// SIMATIC S7-200 project (STEP 7-Micro/WIN), CPU 226 REL 02.00

SYMBOL_TABLE USR1
d1               VD100    // Paper Core
HC               VD0      // Hi Speed Count
HCA              VD150    // Mill Roll Hi speed counter O.S
HCB              VD160    // Mill Roll Hi speed counter D.S
D                VD104    // Diameter
D2               VD108    // Diameter Limit
OUT              VD4      // Hi Speed Count Value
nip              VD112    // Nip
L                VD130    // Web Width
A                VD138    // Nip Setting
nipd             VD116    // Nip display
P                VD120    // Hydraulic press
V                VD204    // Analog out put
DC               AQW0     // 0-10VDC
S3               I0.2     // Paper to lead
S6               I0.5     // Rider roll slow up limit
S9               I1.0     // Lower cradle up limit
S10              I1.1     // Lower cradle down limit
S11              I1.2     // Lower cradle slow down limit
S12              I1.3     // Core chuck (D)
S13              I1.4     // Core chuck p.sw
CS1              I1.5     // Hydraulic pump
PB1              I1.6     // Hydraulic pump on
PB2              I1.7     // Hydraulic pump off
PB3              I2.0     // Trim removal fan ON
PB4              I2.1     // Trim removal fan OFF
PB5              I2.2     // Roll enjctor eject
PB6              I2.3     // Roll ejector return
PB7              I2.4     // Lead roll ON
PB8              I2.5     // Lead roll OFF
PB9              I2.6     // Web tail up
PB10             I2.7     // Web tail down
PB11             I3.0     // Core chuck lift up
PB12             I3.1     // Core chuck lift work
PB13             I3.2     // Core chuck lift down
PB14             I3.3     // Core chuck load
PB15             I3.4     // Core chuck open
PB16             I3.5     // Rder roll up
PB17             I3.6     // Rider roll work
PB18             I3.7     // Rder roll down
PB19             I4.0     // Lower cradle up
PB20             I4.1     // Lower cradle down
PB21             I4.2     // Clutch close
PB22             I4.3     // Auto roll ejector
PB23             I4.4     // Unwinder roll hold
PB24             I4.5     // Unwinder roll release
SP7              I4.6     // sp
SP8              I4.7     // sp
PB27             I5.0     // Lead roll up
PB28             I5.1     // Lead roll down
S14              I5.2     // Water Sensor(oper.side)
S15              I5.3     // Water Sensor(driver.side)
S16              I5.4     // Clutch open limit
S17              I5.5     // Clutch close limit
PB29             I5.6     // Crawl ON
PB30             I5.7     // Crawl  OFF
PB31             I6.0     // Trim ON
PB32             I6.1     // Trim OFF
PB33             I6.2     // Slitter ON
PB34             I6.3     // Slitter OFF
PB35             I6.4     // Blow ON
PB36             I6.5     // Blow OFF
OL1              I6.6     // Trim removal fan OL
OL2A             I6.7     // Hydraulic pump A OL
OL2B             I7.0     // Hydraulic pump B OL
OL3              I7.1     // Lead roll OL
EMG              I7.2     // Emergency
S18              I7.3     // Roll ejector middle limit
ABB1             I7.4     // TOSHIBA RUN
ABB2             I7.5     // TOSHIBA 0 speed
ABB3             I7.6     // TOSHIBA crawl
ABB4             I7.7     // TOSHIBA fault
ABB5             I8.0     // TOSHIBA unwinder brake
ABB6             I8.1     // TOSHIBA lead roll brake
ABB7             I8.2     // TOSHIBA drum brake
ABB8             I8.3     // TOSHIBA warning
S1               I8.4     // Roll ejector forware limit
S2               I8.5     // Roll ejector backware limit
S19              I8.6     // Lead roll motor up limit
S20              I8.7     // Lead roll motor down limit
S13A             I9.0     // Core chuck backward limit
SP4              I9.1     // Mill Roll up-down Motor Over Load O.S
SP5              I9.2     // Mill Roll up-down Motor Over Load D.S
OL8              I9.3     // Mill Roll Move Motor Over Load O.S
S23              I9.4     // Sheed cutter forward limit
S24              I9.5     // Sheed cutter backward limit
S25              I9.6     // Safety hook (D)
S26              I9.7     // Safety hook (O)
PB37             I10.0    // Sheed cutter forward
PB38             I10.1    // Sheed cutter backward
S4               I10.2    // Paper to lead up limit
S5               I10.3    // Rider roll up limit
S7               I10.4    // Rider roll slow down photo
S8               I10.5    // Lower cradle up limit
PB46             I10.6    // Sheed hold
OL9              I10.7    // Mill Roll Move Motor Over Load D.S
PB50             I11.0    // Mill Roll Stand Sync. raise relay
PB51             I11.1    // Mill Roll Stand Sync. lower relay
PB52             I11.2    // Mill Roll move <==  <==
PB53             I11.3    // Mill Roll move ==>  ==>
PB54             I11.4    // Mill Roll move <==  ==>
PB55             I11.5    // Mill Roll move ==>  <==
SP2              I11.6    // UW A or UW B
SP3              I11.7    // sp
S40              I12.0    // Mill Roll Stand raise limits O.S
S41              I12.1    // Mill Roll Stand adj. sensor O.S
S42              I12.2    // Mill Roll stand low limits
S43              I12.3    // Mill Roll Stand raise limits D.S
S44              I12.4    // Mill Roll Stand adj. sensor D.S
S45              I12.5    // Mill Roll Stand down D.S
S46              I12.6    // Mill Roll Move left limits
S47              I12.7    // Mill Roll Move right limits
CR1              Q0.0     // Roll ejector forward valve
CR2              Q0.1     // Roll ejector backward valve
CR3              Q0.2     // Lead roll
CR4              Q0.3     // Paper to lead valve
CR5              Q0.4     // Rider roll up
CR6              Q0.5     // Rider roll fast up
CR7              Q0.6     // Rider roll down
CR8              Q0.7     // Rider roll fast down
CR9              Q1.0     // Rider roll work
CR10             Q1.1     // Alarm buzzer (Rider roll down)
CR11             Q1.2     // Lower cradle up valve
CR12             Q1.3     // Lower cradle fast up valve
CR13             Q1.4     // Lower cradle iccrease press up valve
CR14             Q1.5     // Lower cradle down valve
CR15             Q1.6     // Lower cradle fast down valve
CR16             Q1.7     // Lower cradle down jam valve
CR17             Q2.0     // Lead roll brake
CR18             Q2.1     // Core chuck load
CR19             Q2.2     // Core chuck open
CR20             Q2.3     // Core chuck iccrease press
MCS1             Q2.4     // Trim fan start
MCD1             Q2.5     // Trim fan run
MC2A             Q2.6     // Hydraulic pump A
MC2B             Q2.7     // Hydraulic pump B
CR21             Q3.0     // Buzzer
CR22             Q3.1     // Core chuck lift up
CR23             Q3.2     // Core chuck lift work
CR24             Q3.3     // Paper clip
CR25             Q3.4     // Paper cutter valve
CR26             Q3.5     // Safety hook
PLR1             Q3.6     // Hydraulic pump lamp
PLR2             Q3.7     // Trim removal fan lamp
CR27             Q4.0     // Triming
CR28             Q4.1     // Slitting
CR29             Q4.2     // Blow
CR30             Q4.3     // Clutch valve
CR31             Q4.4     // Unwinder brake valve
CR32             Q4.5     // Drum brake
CR33             Q4.6     // Unwinder roll hold
CR34             Q4.7     // Unwinder roll release
CR35             Q5.0     // sp
CR36             Q5.1     // sp
MCF3             Q5.2     // Lead roll up
MCR3             Q5.3     // Lead roll down
PLR3             Q5.4     // Core chuck load lamp
PLR4             Q5.5     // Rider roll work lamp
PLR5             Q5.6     // Paper clip lamp
PLR6             Q5.7     // sp
CR37             Q6.0     // Ready
CR38             Q6.1     // ABB crawl
CR39             Q6.2     // TOSHIBA Rider Roll Down
CR40             Q6.3     // TOSHIBA roll ejected
CR41             Q6.4     // Clutch valve
CR42             Q6.5     // sp
CR43             Q6.6     // sp
CR44             Q6.7     // sp
CR45             Q7.0     // Sheed cutter forward valve
CR46             Q7.1     // Sheed cutter backward valve
CR47             Q7.2     // sp
CR48             Q7.3     // sp
CR49             Q7.4     // sp
CR50             Q7.5     // sp
MCS              Q7.6     // sp
MCD              Q7.7     // sp
CR51             Q8.0     // Mill Roll Stand Up O.S
CR52             Q8.1     // Mill Roll Stand down O.S
CR53             Q8.2     // Mill Roll Stand Up D.S
CR54             Q8.3     // Mill Roll Stand down D.S
SSP5             Q8.4     // Mill Roll Move Motor left relay O.S
SSP6             Q8.5     // Mill Roll Move Motor right relay O.S
SSP7             Q8.6     // Mill Roll Move Motor left relay D.S
SSP8             Q8.7     // Mill Roll Move Motor right relay D.S
AUX0             M0.0     // Trim removal fan start
AUX6             M0.6     // Clutch
AUX7             M0.7     // Sheed lead
AUX8             M1.0     // Sheed hold
AUX12            M1.4     // Cutter done
AUX13            M1.5     // Rider roll slow down photo
aux14            M2.0     // Sheed cutter base forward
aux15            M2.1     // Sheed cutter base backward
UP1              V1003.0  // Rider roll up limit
UP2              V1003.1  // Rider roll slow up limit reset
DOWN             V1003.2  // Rider roll down
aux31A           V1003.5  // Safety hook
AUX19            V1100.0  // Roll ejector interlock
aux20            V1100.1  // Diameter <
aux22            V1100.2  // Sheed hold
aux23            V1100.3  // Core chuck load
aux24            V1100.4  // Core chuck lift up
aux25            V1100.5  // Roll ejector forward
aux26            V1100.6  // Sheed cutter forward
aux27            V1100.7  // Sheed cutter base backward
aux28            V1102.0  // Roll ejector forward
aux29            V1102.1  // Roll ejector backward delay
aux30            V1102.2  // Roll ejector backward
aux46            V1102.3  // Rider roll raiser
aux31            V1103.1  // O.S value > D.S value
aux32            V1103.2  // O.S value = D.S value
aux33            V1103.3  // O.S value < D.S value
aux34            V1103.4  // Mill Roll Stand Sync. raise
aux35            V1103.5  // Mill Roll Stand Sync. lower
aux36            V1104.0  // Mill Roll move <==  <==
aux37            V1104.1  // Mill Roll move ==>  ==>
aux38            V1104.2  // Mill Roll move <==  ==>
aux39            V1104.3  // Mill Roll move ==>  <==
DOWN2            V1003.4  // Rider roll down
run              V1005.6  // TOSHIBA RUN
UP               V1005.0  // Lower cradle up limit
down3            V1005.2  // Lower cradle down limit
UNWIND           V1101.0  // Clutch
PS               V1020.0  // Press s.w
aux40            V1106.1  // Roll Mill stand single move PB O.S
aux41            V1106.2  // Roll Mill stand single move PB D.S
aux42            V1106.3  // Roll Mill stand Sync. move PB O.S
aux43            V1107.0  // Roll Mill stand single move  O.S
aux44            V1107.1  // Roll Mill stand single move  D.S
aux45            V1107.2  // Roll Mill stand Sync. move
END_SYMBOL_TABLE

ORGANIZATION_BLOCK OB_1:OB1
TITLE= PROGRAM COMMENTS
// Press F1 for help and example program 
BEGIN
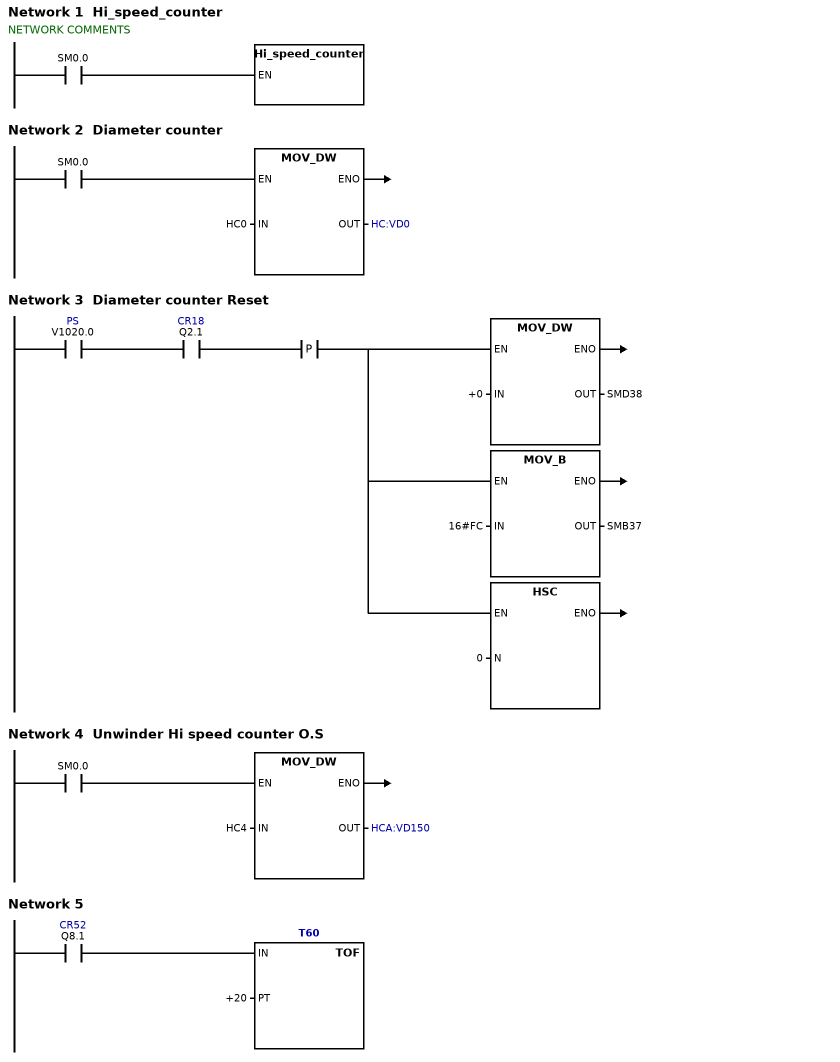
Network 1 // Hi_speed_counter
//  NETWORK COMMENTS
LD     SM0.0
CALL   Hi_speed_counter:SBR1
Network 2 // Diameter counter
LD     SM0.0
MOVD   HC0, HC:VD0
Network 3 // Diameter counter Reset
LD     PS:V1020.0
A      CR18:Q2.1
EU
MOVD   +0, SMD38
MOVB   16#FC, SMB37
HSC    0
Network 4 // Unwinder Hi speed counter O.S
LD     SM0.0
MOVD   HC4, HCA:VD150
Network 5
LD     CR52:Q8.1
TOF    T60, +20
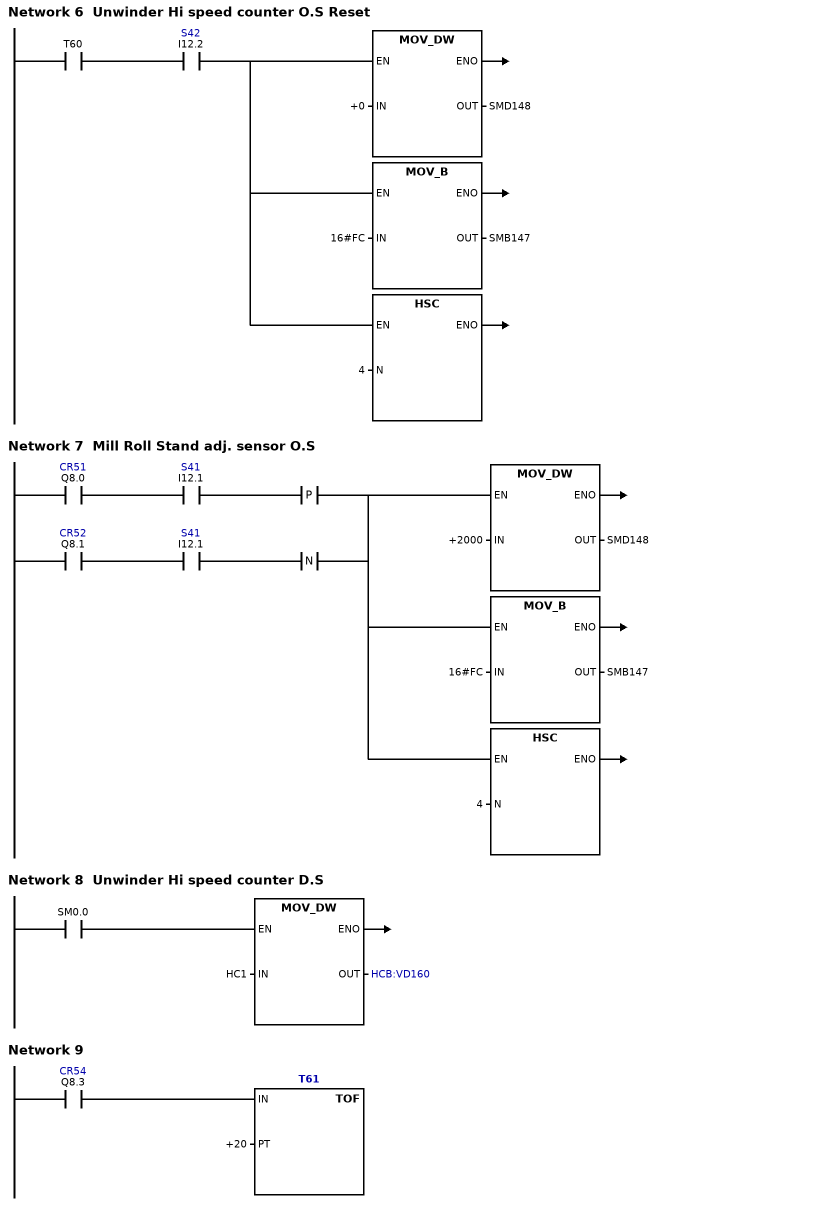
Network 6 // Unwinder Hi speed counter O.S Reset
LD     T60
A      S42:I12.2
MOVD   +0, SMD148
MOVB   16#FC, SMB147
HSC    4
Network 7 // Mill Roll Stand adj. sensor O.S
LD     CR51:Q8.0
A      S41:I12.1
EU
LD     CR52:Q8.1
A      S41:I12.1
ED
OLD
MOVD   +2000, SMD148
MOVB   16#FC, SMB147
HSC    4
Network 8 // Unwinder Hi speed counter D.S
LD     SM0.0
MOVD   HC1, HCB:VD160
Network 9
LD     CR54:Q8.3
TOF    T61, +20
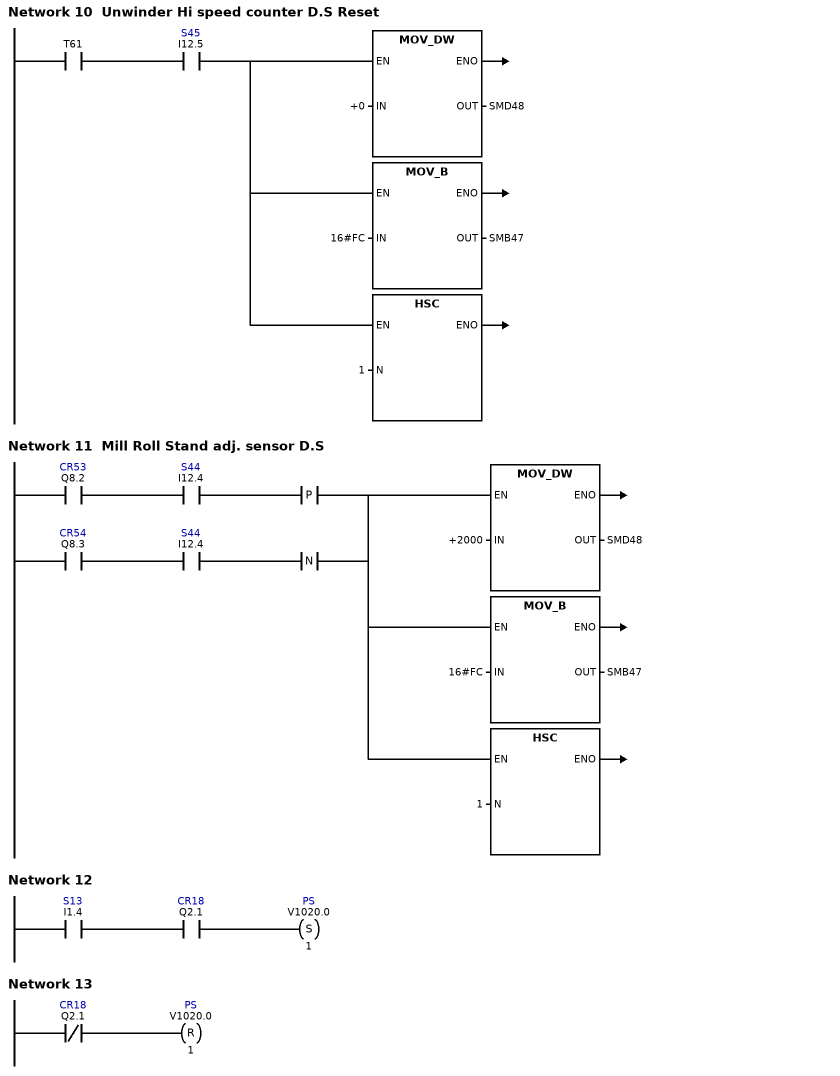
Network 10 // Unwinder Hi speed counter D.S Reset
LD     T61
A      S45:I12.5
MOVD   +0, SMD48
MOVB   16#FC, SMB47
HSC    1
Network 11 // Mill Roll Stand adj. sensor D.S
LD     CR53:Q8.2
A      S44:I12.4
EU
LD     CR54:Q8.3
A      S44:I12.4
ED
OLD
MOVD   +2000, SMD48
MOVB   16#FC, SMB47
HSC    1
Network 12
LD     S13:I1.4
A      CR18:Q2.1
S      PS:V1020.0, 1
Network 13
LDN    CR18:Q2.1
R      PS:V1020.0, 1
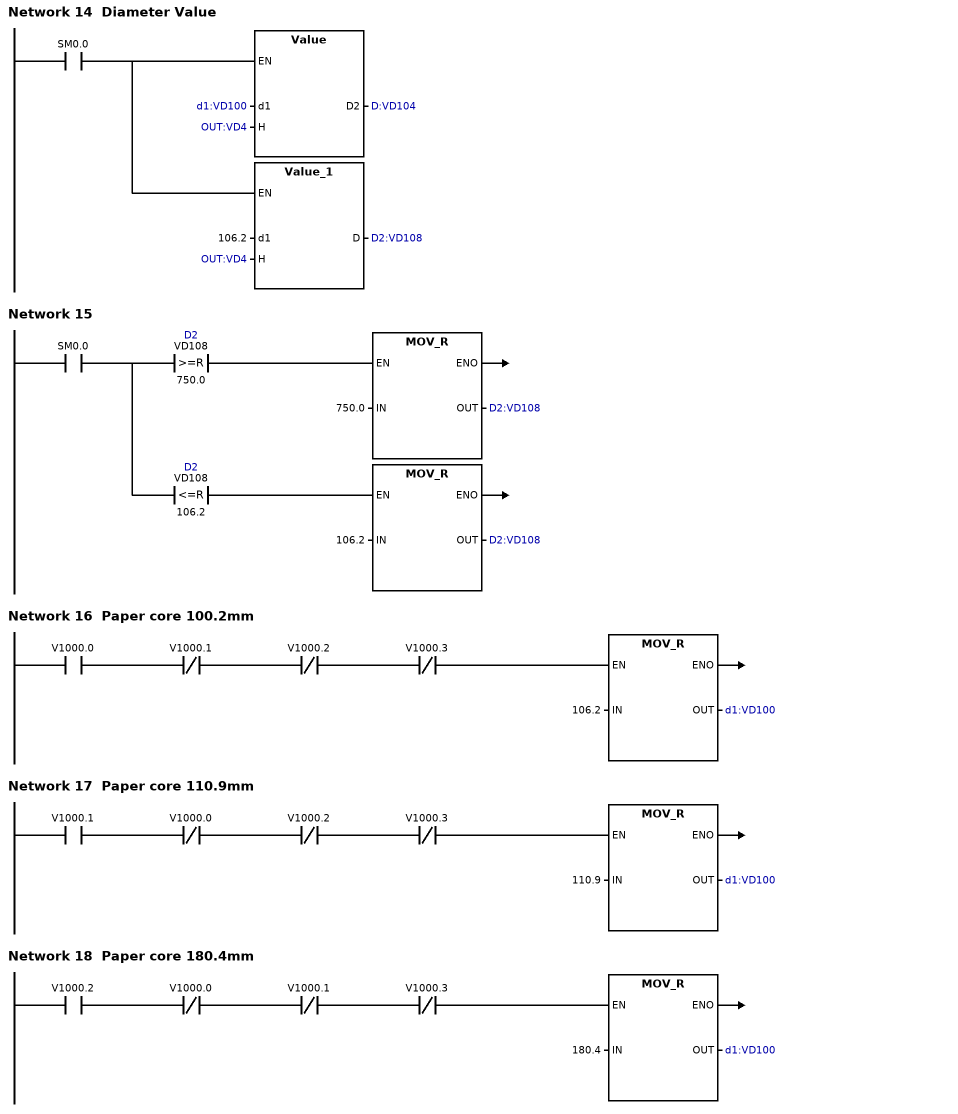
Network 14 // Diameter Value
LD     SM0.0
CALL   Value:SBR0, d1:VD100, OUT:VD4, D:VD104
CALL   Value_1:SBR10, 106.2, OUT:VD4, D2:VD108
Network 15
LD     SM0.0
LPS
AR>=   D2:VD108, 750.0
MOVR   750.0, D2:VD108
LPP
AR<=   D2:VD108, 106.2
MOVR   106.2, D2:VD108
Network 16 // Paper core 100.2mm
LD     V1000.0
AN     V1000.1
AN     V1000.2
AN     V1000.3
MOVR   106.2, d1:VD100
Network 17 // Paper core 110.9mm
LD     V1000.1
AN     V1000.0
AN     V1000.2
AN     V1000.3
MOVR   110.9, d1:VD100
Network 18 // Paper core 180.4mm
LD     V1000.2
AN     V1000.0
AN     V1000.1
AN     V1000.3
MOVR   180.4, d1:VD100
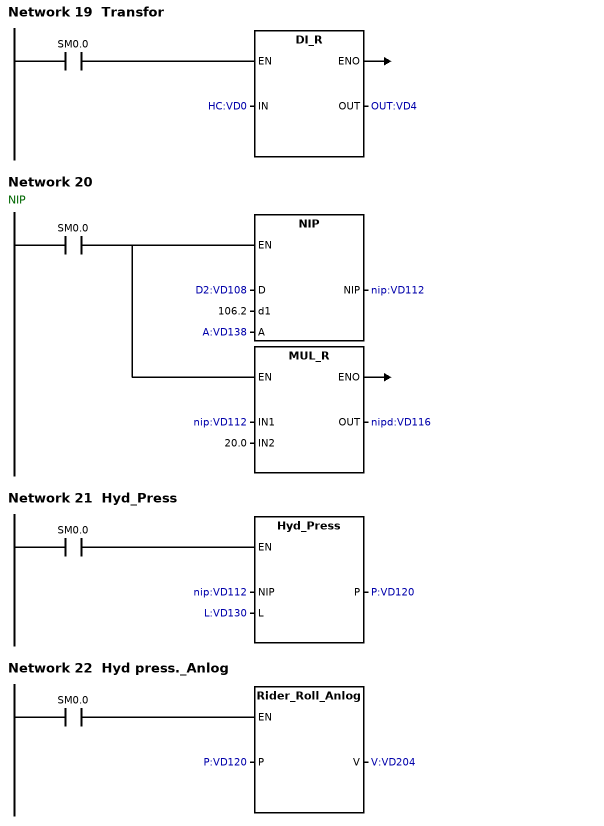
Network 19 // Transfor
LD     SM0.0
DTR    HC:VD0, OUT:VD4
Network 20
// NIP
LD     SM0.0
CALL   NIP:SBR2, D2:VD108, 106.2, A:VD138, nip:VD112
MOVR   nip:VD112, nipd:VD116
*R     20.0, nipd:VD116
Network 21 // Hyd_Press
LD     SM0.0
CALL   Hyd_Press:SBR3, nip:VD112, L:VD130, P:VD120
Network 22 // Hyd press._Anlog
LD     SM0.0
CALL   Rider_Roll_Anlog:SBR4, P:VD120, V:VD204
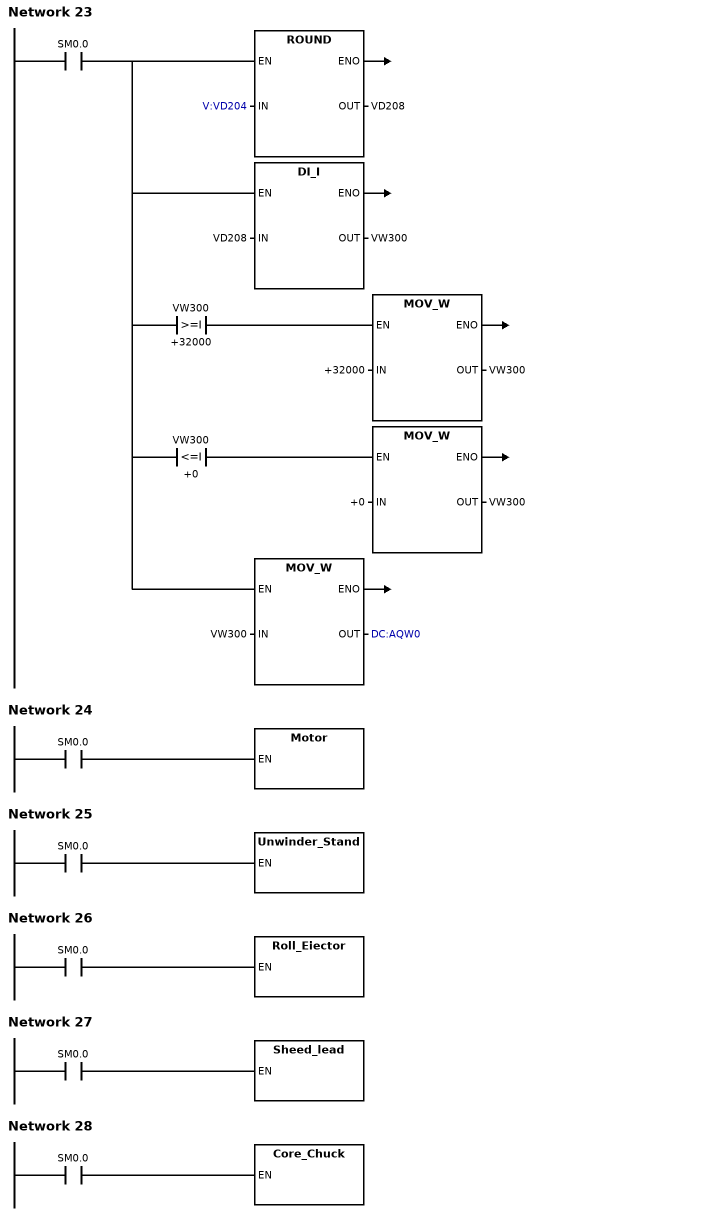
Network 23
LD     SM0.0
LPS
ROUND  V:VD204, VD208
DTI    VD208, VW300
AW>=   VW300, +32000
MOVW   +32000, VW300
LRD
AW<=   VW300, +0
MOVW   +0, VW300
LPP
MOVW   VW300, DC:AQW0
Network 24
LD     SM0.0
CALL   Motor:SBR5
Network 25
LD     SM0.0
CALL   Unwinder_Stand:SBR6
Network 26
LD     SM0.0
CALL   Roll_Eiector:SBR7
Network 27
LD     SM0.0
CALL   Sheed_lead:SBR8
Network 28
LD     SM0.0
CALL   Core_Chuck:SBR9
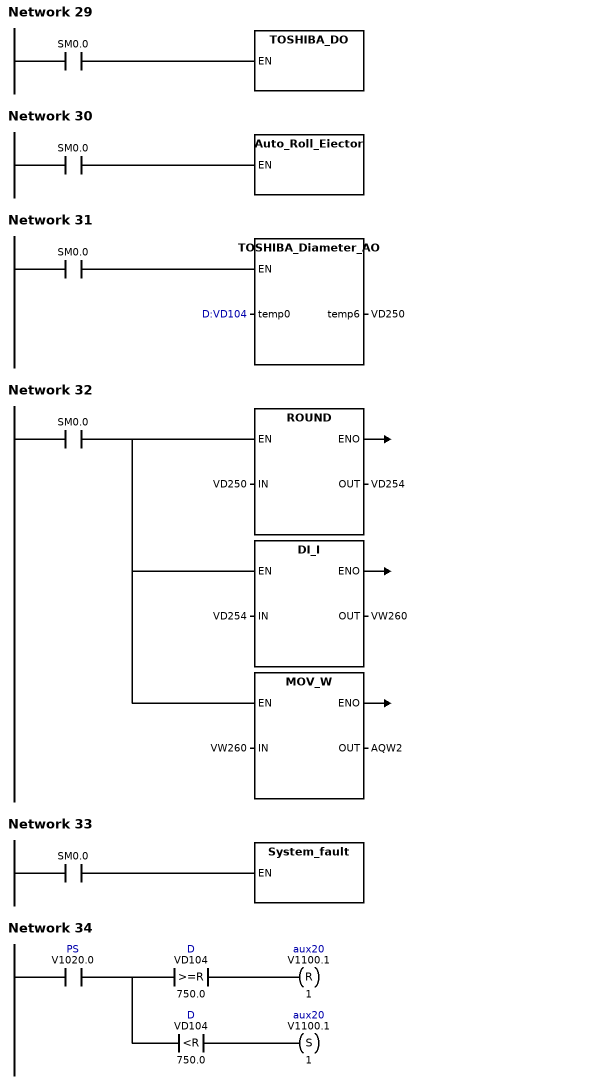
Network 29
LD     SM0.0
CALL   TOSHIBA_DO:SBR11
Network 30
LD     SM0.0
CALL   Auto_Roll_Eiector:SBR12
Network 31
LD     SM0.0
CALL   TOSHIBA_Diameter_AO:SBR13, D:VD104, VD250
Network 32
LD     SM0.0
ROUND  VD250, VD254
DTI    VD254, VW260
MOVW   VW260, AQW2
Network 33
LD     SM0.0
CALL   System_fault:SBR14
Network 34
LD     PS:V1020.0
LPS
AR>=   D:VD104, 750.0
R      aux20:V1100.1, 1
LPP
AR<    D:VD104, 750.0
S      aux20:V1100.1, 1
END_ORGANIZATION_BLOCK

SUBROUTINE_BLOCK Value:SBR0
TITLE= SUBROUTINE COMMENTS
// Press F1 for help and example program 
VAR_INPUT
d1:REAL;	// LD0 
H:REAL;	// LD4 
END_VAR
VAR_OUTPUT
D2:REAL;	// LD8 
END_VAR
VAR
TEMP1:REAL;	// LD12 
TEMP2:REAL;	// LD16 
TEMP3:REAL;	// LD20 
TEMP4:REAL;	// LD24 
TEMP5:REAL;	// LD28 
TEMP6:REAL;	// LD32 
TEMP7:REAL;	// LD36 
TEMP8:REAL;	// LD40 
TEMP9:REAL;	// LD44 
TEMP10:REAL;	// LD48 
TEMP11:REAL;	// LD52 
END_VAR
BEGIN
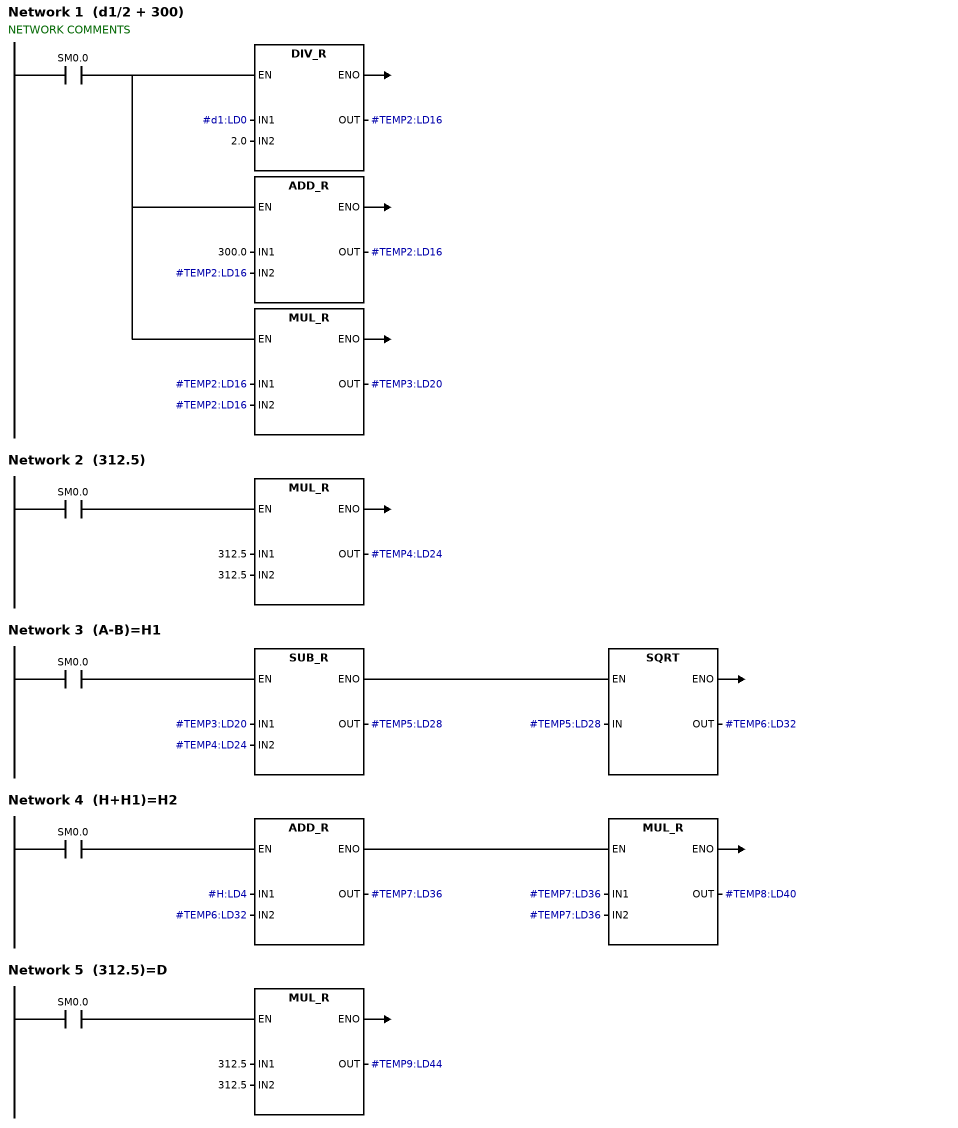
Network 1 // (d1/2 + 300)
//  NETWORK COMMENTS
LD     SM0.0
MOVR   #d1:LD0, #TEMP2:LD16
/R     2.0, #TEMP2:LD16
+R     300.0, #TEMP2:LD16
MOVR   #TEMP2:LD16, #TEMP3:LD20
*R     #TEMP2:LD16, #TEMP3:LD20
Network 2 // (312.5)
LD     SM0.0
MOVR   312.5, #TEMP4:LD24
*R     312.5, #TEMP4:LD24
Network 3 // (A-B)=H1
LD     SM0.0
MOVR   #TEMP3:LD20, #TEMP5:LD28
AENO
-R     #TEMP4:LD24, #TEMP5:LD28
AENO
SQRT   #TEMP5:LD28, #TEMP6:LD32
Network 4 // (H+H1)=H2
LD     SM0.0
MOVR   #H:LD4, #TEMP7:LD36
AENO
+R     #TEMP6:LD32, #TEMP7:LD36
AENO
MOVR   #TEMP7:LD36, #TEMP8:LD40
*R     #TEMP7:LD36, #TEMP8:LD40
Network 5 // (312.5)=D
LD     SM0.0
MOVR   312.5, #TEMP9:LD44
*R     312.5, #TEMP9:LD44
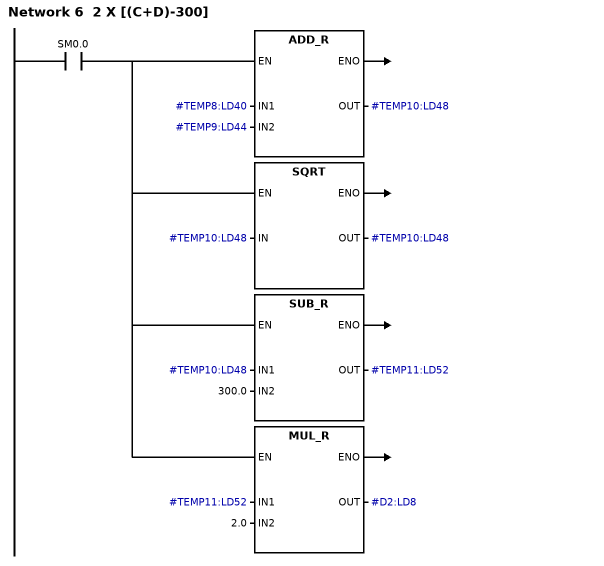
Network 6 // 2 X [(C+D)-300]
LD     SM0.0
MOVR   #TEMP8:LD40, #TEMP10:LD48
+R     #TEMP9:LD44, #TEMP10:LD48
SQRT   #TEMP10:LD48, #TEMP10:LD48
MOVR   #TEMP10:LD48, #TEMP11:LD52
-R     300.0, #TEMP11:LD52
MOVR   #TEMP11:LD52, #D2:LD8
*R     2.0, #D2:LD8
END_SUBROUTINE_BLOCK

SUBROUTINE_BLOCK Hi_speed_counter:SBR1
TITLE=This POU was created by the HSC formula of the S7-200 Instruction Wizard.
// This Subroutine configures HC0 for Mode 9 operation.  It contains initialization code and attaches the Interrupt Routines created by the wizard.  To enable this configuration within the program, Use SM0.1 or an edge-triggered instruction to call this Subroutine once from the MAIN program block.  
BEGIN
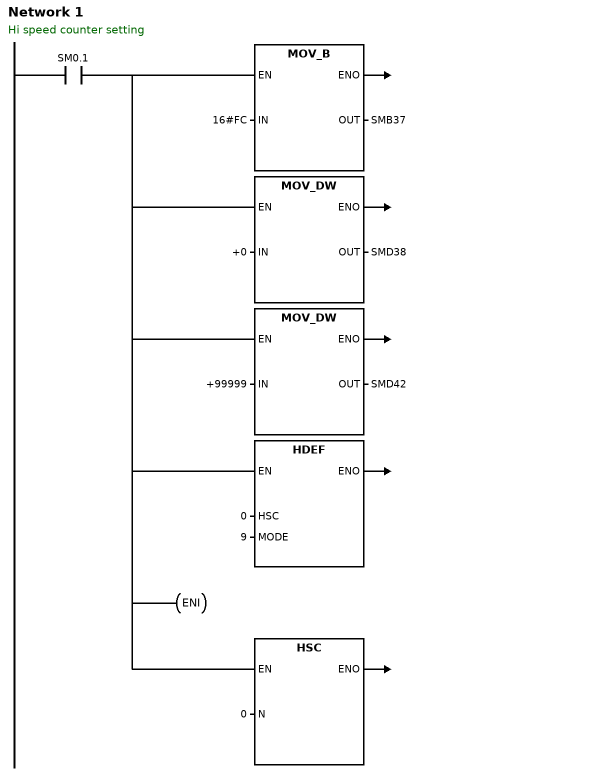
Network 1 //   
// Hi speed counter setting
//Set control bits: count UP; rate 1X; enabled; 
//CV = 0; 
//PV = 0; 
LD     SM0.1
MOVB   16#FC, SMB37
MOVD   +0, SMD38
MOVD   +99999, SMD42
HDEF   0, 9
ENI
HSC    0
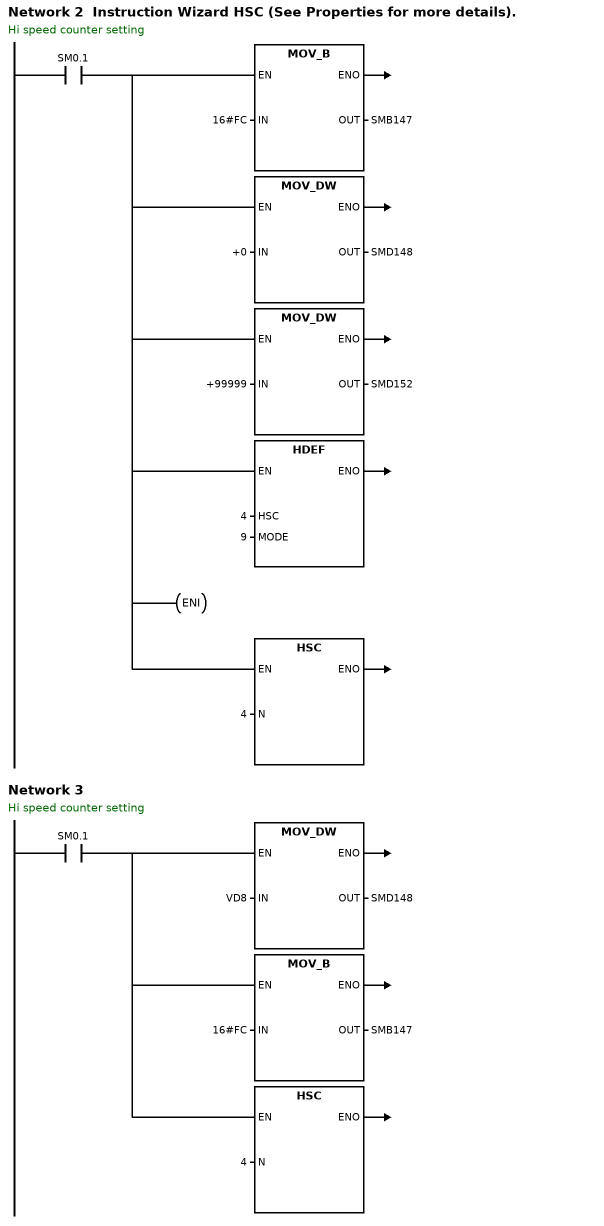
Network 2 // Instruction Wizard HSC (See Properties for more details).  
// Hi speed counter setting
//Set control bits: count UP; rate 1X; enabled; 
//CV = 0; 
//PV = 0; 
LD     SM0.1
MOVB   16#FC, SMB147
MOVD   +0, SMD148
MOVD   +99999, SMD152
HDEF   4, 9
ENI
HSC    4
Network 3
// Hi speed counter setting
LD     SM0.1
MOVD   VD8, SMD148
MOVB   16#FC, SMB147
HSC    4
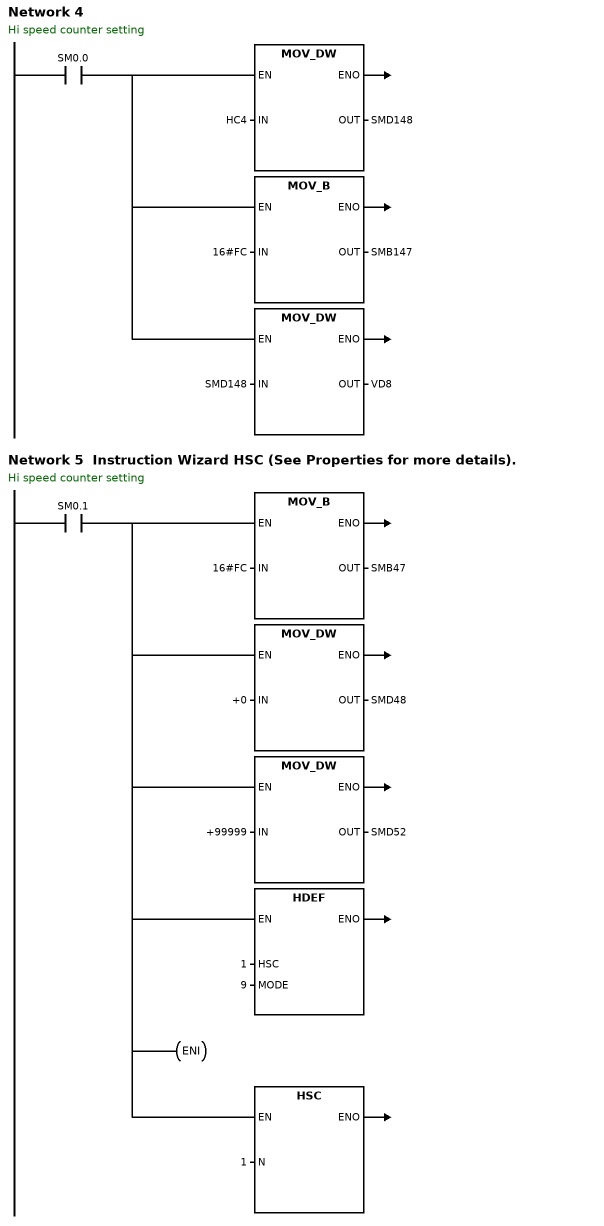
Network 4
// Hi speed counter setting
LD     SM0.0
MOVD   HC4, SMD148
MOVB   16#FC, SMB147
MOVD   SMD148, VD8
Network 5 // Instruction Wizard HSC (See Properties for more details).  
// Hi speed counter setting
//Set control bits: count UP; rate 1X; enabled; 
//CV = 0; 
//PV = 0; 
LD     SM0.1
MOVB   16#FC, SMB47
MOVD   +0, SMD48
MOVD   +99999, SMD52
HDEF   1, 9
ENI
HSC    1
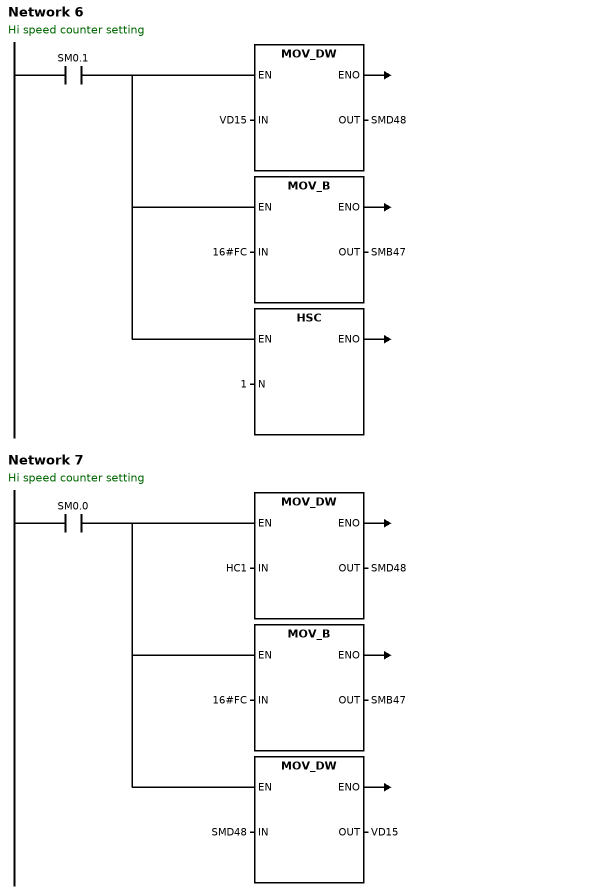
Network 6
// Hi speed counter setting
LD     SM0.1
MOVD   VD15, SMD48
MOVB   16#FC, SMB47
HSC    1
Network 7
// Hi speed counter setting
LD     SM0.0
MOVD   HC1, SMD48
MOVB   16#FC, SMB47
MOVD   SMD48, VD15
END_SUBROUTINE_BLOCK

SUBROUTINE_BLOCK NIP:SBR2
TITLE= SUBROUTINE COMMENTS
// Press F1 for help and example program 
VAR_INPUT
D:REAL;	// LD0 
d1:REAL;	// LD4 
A:REAL;	// LD8 
END_VAR
VAR_OUTPUT
NIP:REAL;	// LD12 
END_VAR
VAR
TEMP1:REAL;	// LD16 
TEMP2:REAL;	// LD20 
TEMP3:REAL;	// LD24 
TEMP4:REAL;	// LD28 
TEMP5:REAL;	// LD32 
TEMP6:REAL;	// LD36 
TEMP7:REAL;	// LD40 
END_VAR
BEGIN
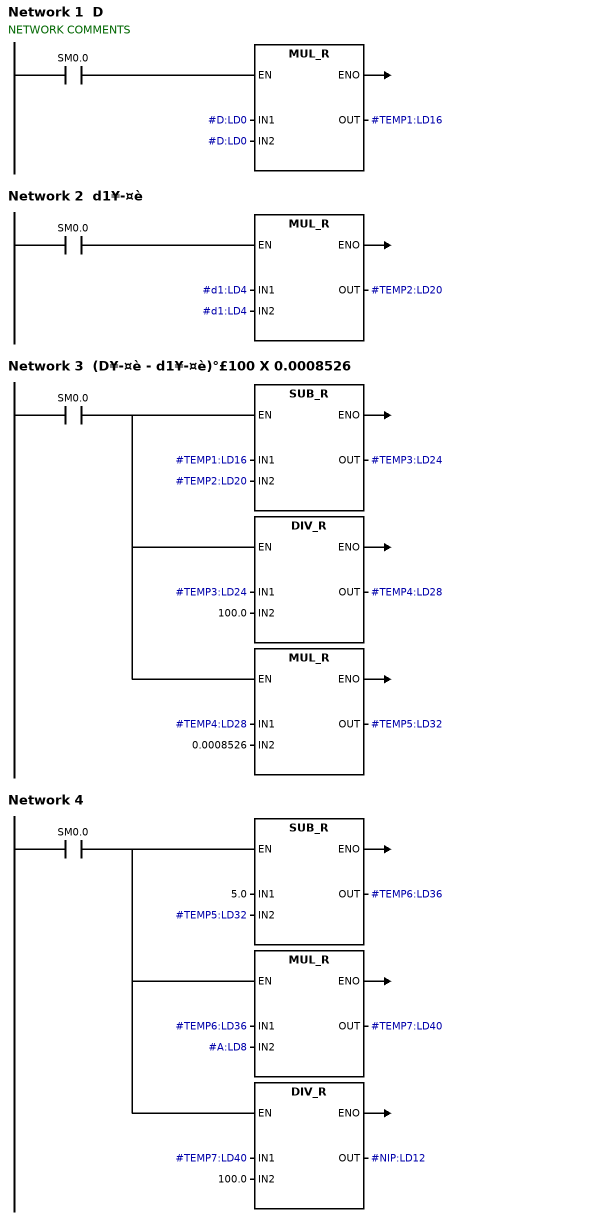
Network 1 // D
//  NETWORK COMMENTS
LD     SM0.0
MOVR   #D:LD0, #TEMP1:LD16
*R     #D:LD0, #TEMP1:LD16
Network 2 // d1平方
LD     SM0.0
MOVR   #d1:LD4, #TEMP2:LD20
*R     #d1:LD4, #TEMP2:LD20
Network 3 // (D平方 - d1平方)除100 X 0.0008526
LD     SM0.0
MOVR   #TEMP1:LD16, #TEMP3:LD24
-R     #TEMP2:LD20, #TEMP3:LD24
MOVR   #TEMP3:LD24, #TEMP4:LD28
/R     100.0, #TEMP4:LD28
MOVR   #TEMP4:LD28, #TEMP5:LD32
*R     0.0008526, #TEMP5:LD32
Network 4
LD     SM0.0
MOVR   5.0, #TEMP6:LD36
-R     #TEMP5:LD32, #TEMP6:LD36
MOVR   #TEMP6:LD36, #TEMP7:LD40
*R     #A:LD8, #TEMP7:LD40
MOVR   #TEMP7:LD40, #NIP:LD12
/R     100.0, #NIP:LD12
END_SUBROUTINE_BLOCK

SUBROUTINE_BLOCK Hyd_Press:SBR3
TITLE= SUBROUTINE COMMENTS
// Press F1 for help and example program 
VAR_INPUT
NIP:REAL;	// LD0 
L:REAL;	// LD4 
END_VAR
VAR_OUTPUT
P:REAL;	// LD8 
END_VAR
VAR
TEMP1:REAL;	// LD12 
TEMP2:REAL;	// LD16 
TEMP3:REAL;	// LD20 
END_VAR
BEGIN
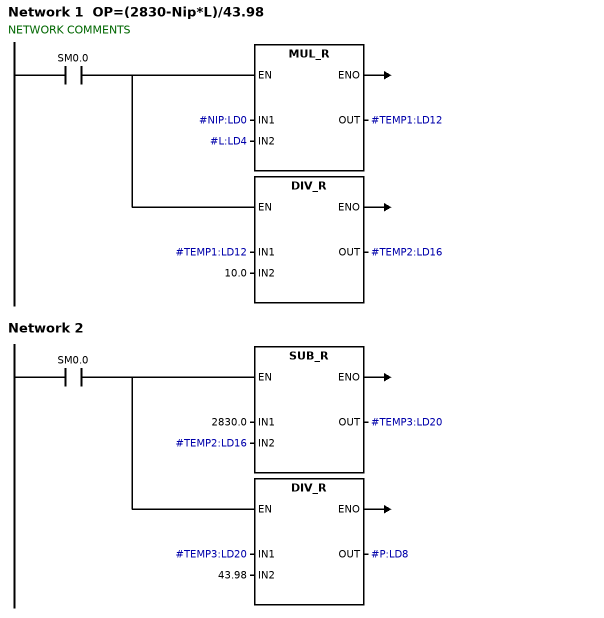
Network 1 // OP=(2830-Nip*L)/43.98
//  NETWORK COMMENTS
LD     SM0.0
MOVR   #NIP:LD0, #TEMP1:LD12
*R     #L:LD4, #TEMP1:LD12
MOVR   #TEMP1:LD12, #TEMP2:LD16
/R     10.0, #TEMP2:LD16
Network 2
LD     SM0.0
MOVR   2830.0, #TEMP3:LD20
-R     #TEMP2:LD16, #TEMP3:LD20
MOVR   #TEMP3:LD20, #P:LD8
/R     43.98, #P:LD8
END_SUBROUTINE_BLOCK

SUBROUTINE_BLOCK Rider_Roll_Anlog:SBR4
TITLE= SUBROUTINE COMMENTS
// Press F1 for help and example program 
VAR_INPUT
P:REAL;	// LD0 
END_VAR
VAR_OUTPUT
V:REAL;	// LD4 
END_VAR
VAR
TEMP1:REAL;	// LD8 
END_VAR
BEGIN
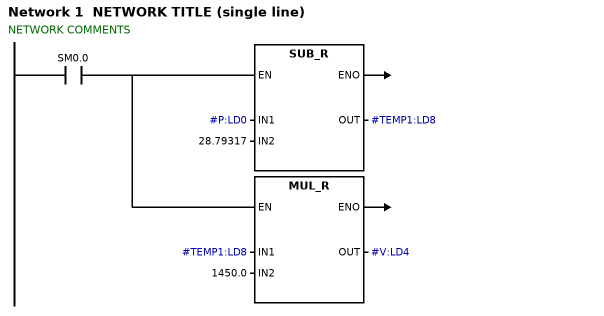
Network 1 // NETWORK TITLE (single line)
//  NETWORK COMMENTS
LD     SM0.0
MOVR   #P:LD0, #TEMP1:LD8
-R     28.79317, #TEMP1:LD8
MOVR   #TEMP1:LD8, #V:LD4
*R     1450.0, #V:LD4
END_SUBROUTINE_BLOCK

SUBROUTINE_BLOCK Motor:SBR5
TITLE= SUBROUTINE COMMENTS
// Press F1 for help and example program 
BEGIN
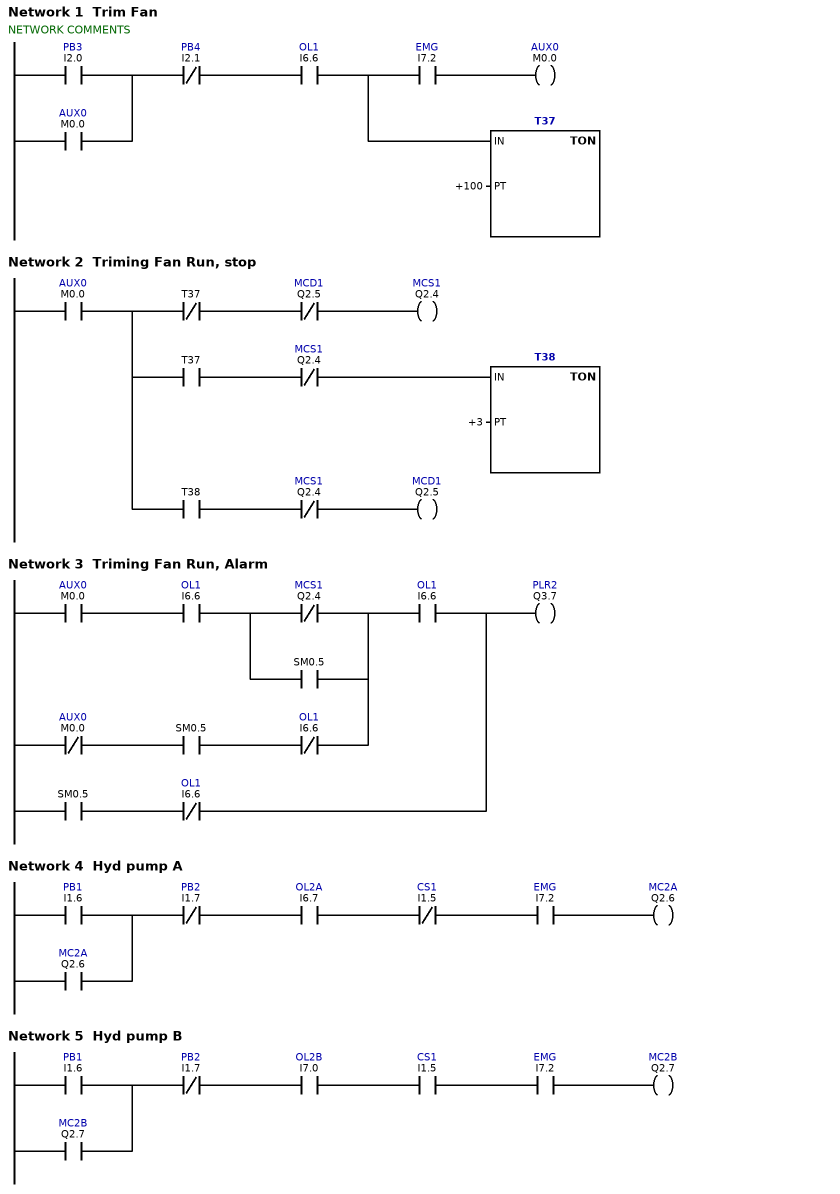
Network 1 // Trim Fan
//  NETWORK COMMENTS
LD     PB3:I2.0
O      AUX0:M0.0
AN     PB4:I2.1
A      OL1:I6.6
LPS
A      EMG:I7.2
=      AUX0:M0.0
LPP
TON    T37, +100
Network 2 // Triming Fan Run, stop
LD     AUX0:M0.0
LPS
AN     T37
AN     MCD1:Q2.5
=      MCS1:Q2.4
LRD
A      T37
AN     MCS1:Q2.4
TON    T38, +3
LPP
A      T38
AN     MCS1:Q2.4
=      MCD1:Q2.5
Network 3 // Triming Fan Run, Alarm
LD     AUX0:M0.0
A      OL1:I6.6
LDN    MCS1:Q2.4
O      SM0.5
ALD
LDN    AUX0:M0.0
A      SM0.5
AN     OL1:I6.6
OLD
A      OL1:I6.6
LD     SM0.5
AN     OL1:I6.6
OLD
=      PLR2:Q3.7
Network 4 // Hyd pump A
LD     PB1:I1.6
O      MC2A:Q2.6
AN     PB2:I1.7
A      OL2A:I6.7
AN     CS1:I1.5
A      EMG:I7.2
=      MC2A:Q2.6
Network 5 // Hyd pump B
LD     PB1:I1.6
O      MC2B:Q2.7
AN     PB2:I1.7
A      OL2B:I7.0
A      CS1:I1.5
A      EMG:I7.2
=      MC2B:Q2.7
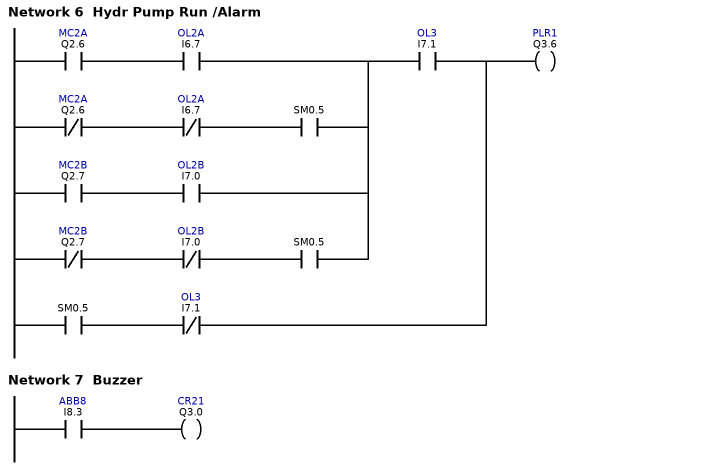
Network 6 // Hydr Pump Run /Alarm
LD     MC2A:Q2.6
A      OL2A:I6.7
LDN    MC2A:Q2.6
AN     OL2A:I6.7
A      SM0.5
OLD
LD     MC2B:Q2.7
A      OL2B:I7.0
OLD
LDN    MC2B:Q2.7
AN     OL2B:I7.0
A      SM0.5
OLD
A      OL3:I7.1
LD     SM0.5
AN     OL3:I7.1
OLD
=      PLR1:Q3.6
Network 7 // Buzzer
LD     ABB8:I8.3
=      CR21:Q3.0
END_SUBROUTINE_BLOCK

SUBROUTINE_BLOCK Unwinder_Stand:SBR6
TITLE= SUBROUTINE COMMENTS
// Press F1 for help and example program 
BEGIN
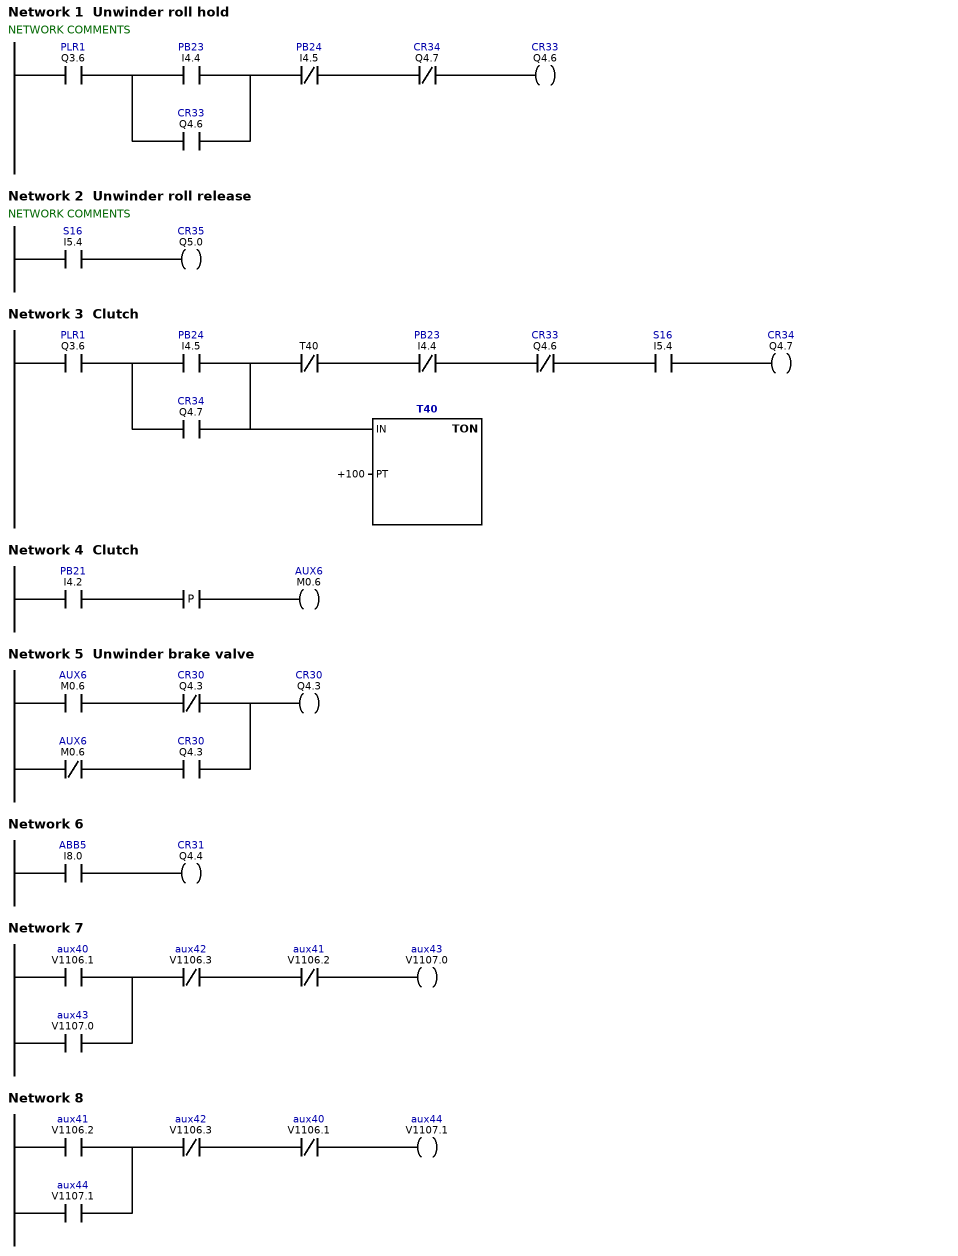
Network 1 // Unwinder roll hold
//  NETWORK COMMENTS
LD     PLR1:Q3.6
LD     PB23:I4.4
O      CR33:Q4.6
ALD
AN     PB24:I4.5
AN     CR34:Q4.7
=      CR33:Q4.6
Network 2 // Unwinder roll release
//  NETWORK COMMENTS
LD     S16:I5.4
=      CR35:Q5.0
Network 3 // Clutch
LD     PLR1:Q3.6
LD     PB24:I4.5
O      CR34:Q4.7
ALD
LPS
AN     T40
AN     PB23:I4.4
AN     CR33:Q4.6
A      S16:I5.4
=      CR34:Q4.7
LPP
TON    T40, +100
Network 4 // Clutch
LD     PB21:I4.2
EU
=      AUX6:M0.6
Network 5 // Unwinder brake valve
LD     AUX6:M0.6
AN     CR30:Q4.3
LDN    AUX6:M0.6
A      CR30:Q4.3
OLD
=      CR30:Q4.3
Network 6
LD     ABB5:I8.0
=      CR31:Q4.4
Network 7
LD     aux40:V1106.1
O      aux43:V1107.0
AN     aux42:V1106.3
AN     aux41:V1106.2
=      aux43:V1107.0
Network 8
LD     aux41:V1106.2
O      aux44:V1107.1
AN     aux42:V1106.3
AN     aux40:V1106.1
=      aux44:V1107.1
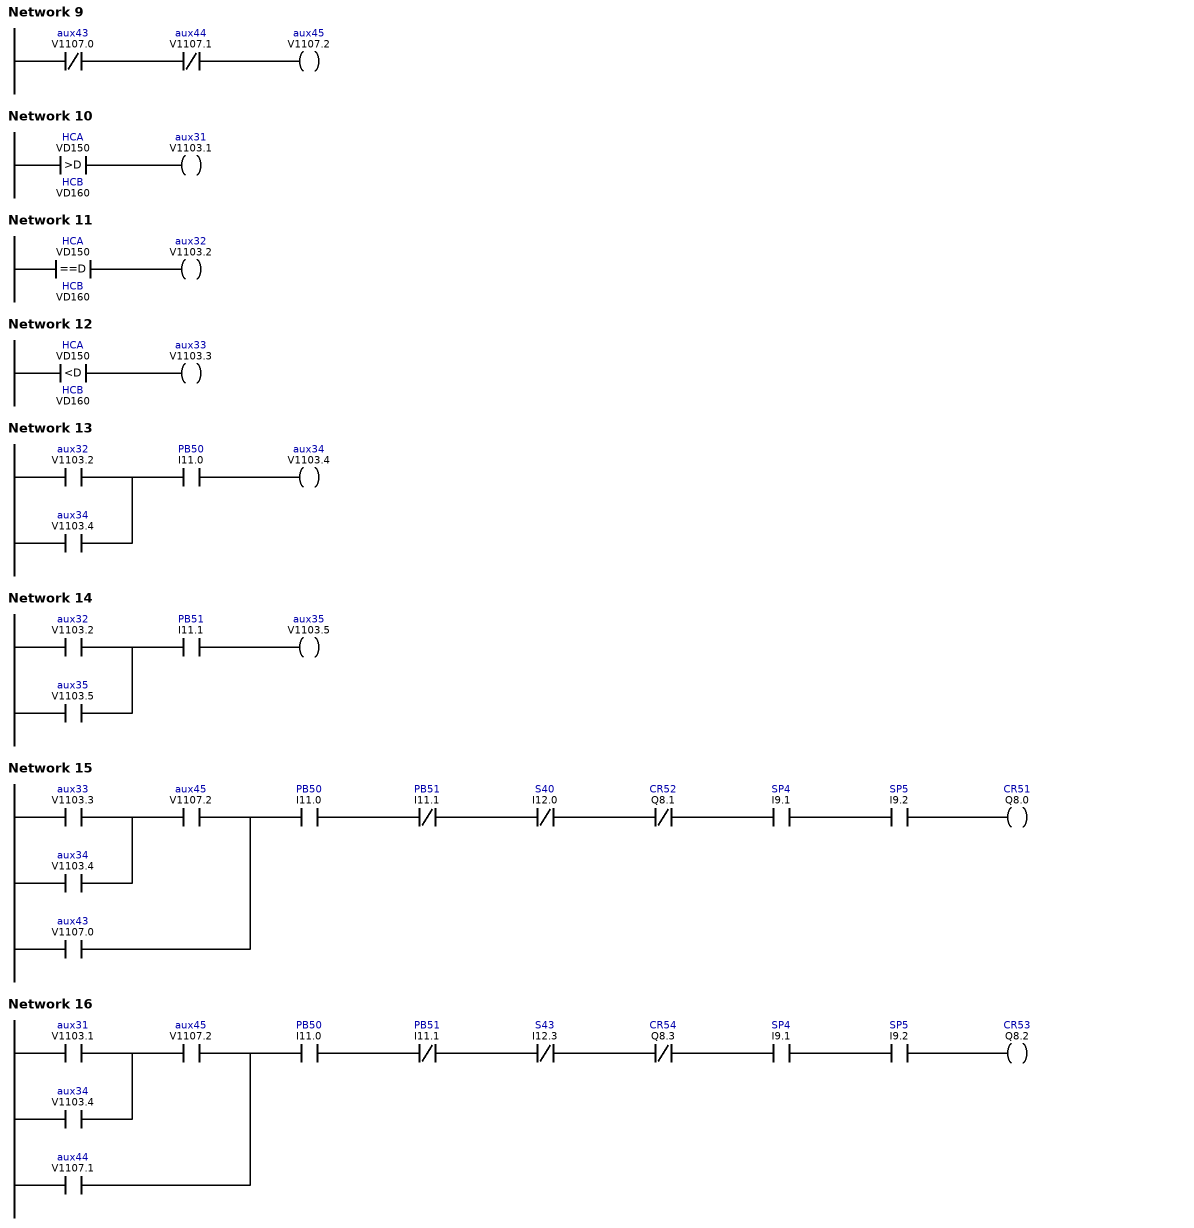
Network 9
LDN    aux43:V1107.0
AN     aux44:V1107.1
=      aux45:V1107.2
Network 10
LDD>   HCA:VD150, HCB:VD160
=      aux31:V1103.1
Network 11
LDD=   HCA:VD150, HCB:VD160
=      aux32:V1103.2
Network 12
LDD<   HCA:VD150, HCB:VD160
=      aux33:V1103.3
Network 13
LD     aux32:V1103.2
O      aux34:V1103.4
A      PB50:I11.0
=      aux34:V1103.4
Network 14
LD     aux32:V1103.2
O      aux35:V1103.5
A      PB51:I11.1
=      aux35:V1103.5
Network 15
LD     aux33:V1103.3
O      aux34:V1103.4
A      aux45:V1107.2
O      aux43:V1107.0
A      PB50:I11.0
AN     PB51:I11.1
AN     S40:I12.0
AN     CR52:Q8.1
A      SP4:I9.1
A      SP5:I9.2
=      CR51:Q8.0
Network 16
LD     aux31:V1103.1
O      aux34:V1103.4
A      aux45:V1107.2
O      aux44:V1107.1
A      PB50:I11.0
AN     PB51:I11.1
AN     S43:I12.3
AN     CR54:Q8.3
A      SP4:I9.1
A      SP5:I9.2
=      CR53:Q8.2
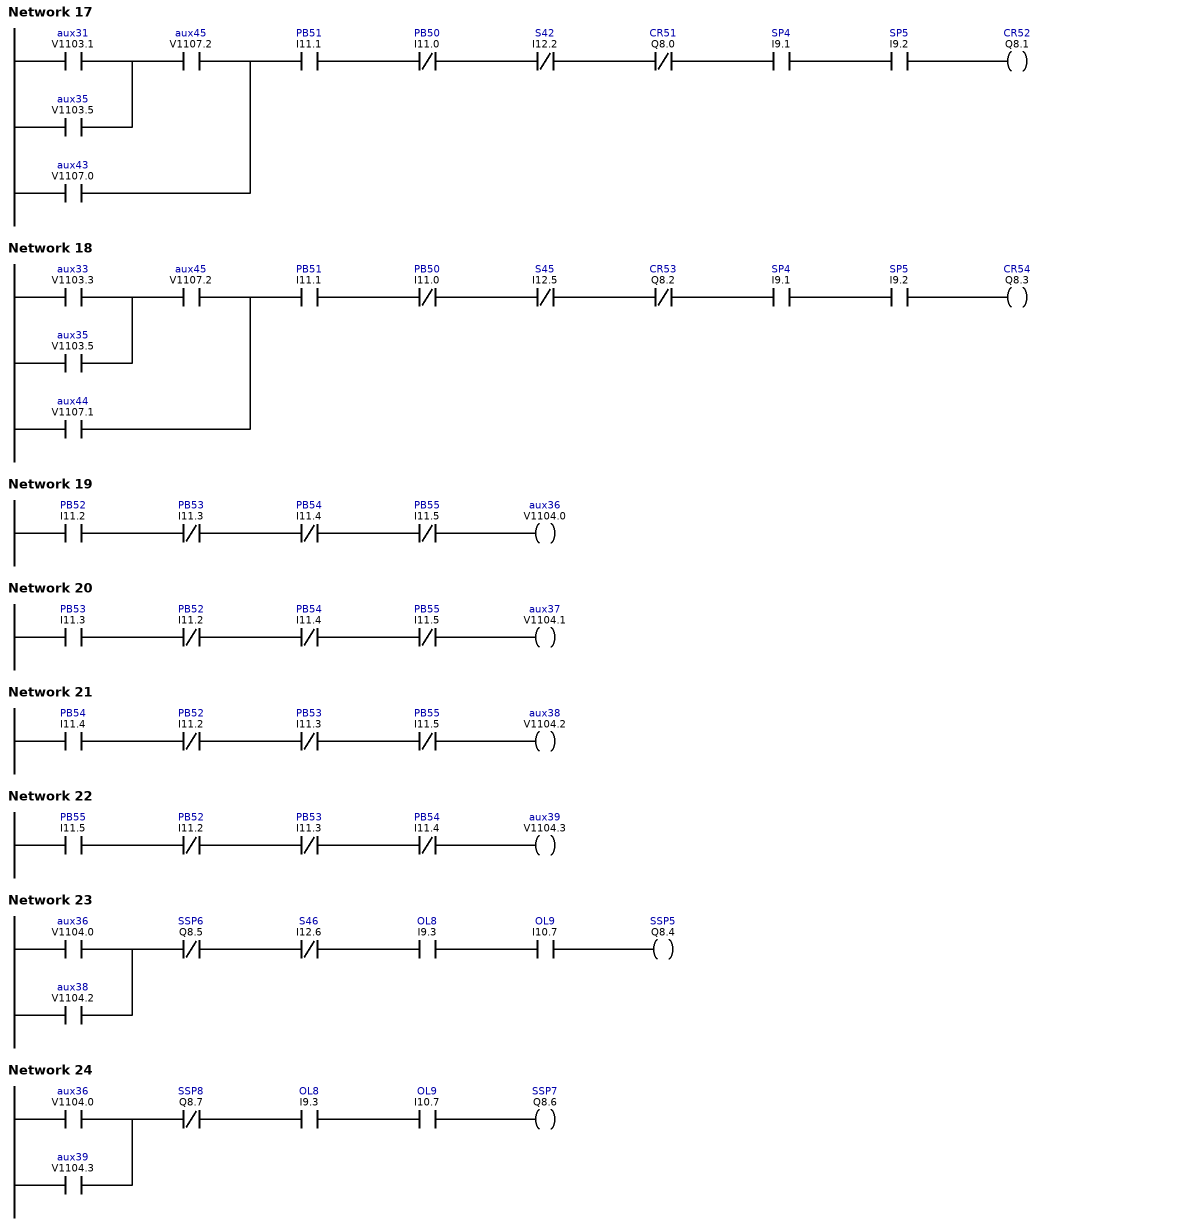
Network 17
LD     aux31:V1103.1
O      aux35:V1103.5
A      aux45:V1107.2
O      aux43:V1107.0
A      PB51:I11.1
AN     PB50:I11.0
AN     S42:I12.2
AN     CR51:Q8.0
A      SP4:I9.1
A      SP5:I9.2
=      CR52:Q8.1
Network 18
LD     aux33:V1103.3
O      aux35:V1103.5
A      aux45:V1107.2
O      aux44:V1107.1
A      PB51:I11.1
AN     PB50:I11.0
AN     S45:I12.5
AN     CR53:Q8.2
A      SP4:I9.1
A      SP5:I9.2
=      CR54:Q8.3
Network 19
LD     PB52:I11.2
AN     PB53:I11.3
AN     PB54:I11.4
AN     PB55:I11.5
=      aux36:V1104.0
Network 20
LD     PB53:I11.3
AN     PB52:I11.2
AN     PB54:I11.4
AN     PB55:I11.5
=      aux37:V1104.1
Network 21
LD     PB54:I11.4
AN     PB52:I11.2
AN     PB53:I11.3
AN     PB55:I11.5
=      aux38:V1104.2
Network 22
LD     PB55:I11.5
AN     PB52:I11.2
AN     PB53:I11.3
AN     PB54:I11.4
=      aux39:V1104.3
Network 23
LD     aux36:V1104.0
O      aux38:V1104.2
AN     SSP6:Q8.5
AN     S46:I12.6
A      OL8:I9.3
A      OL9:I10.7
=      SSP5:Q8.4
Network 24
LD     aux36:V1104.0
O      aux39:V1104.3
AN     SSP8:Q8.7
A      OL8:I9.3
A      OL9:I10.7
=      SSP7:Q8.6
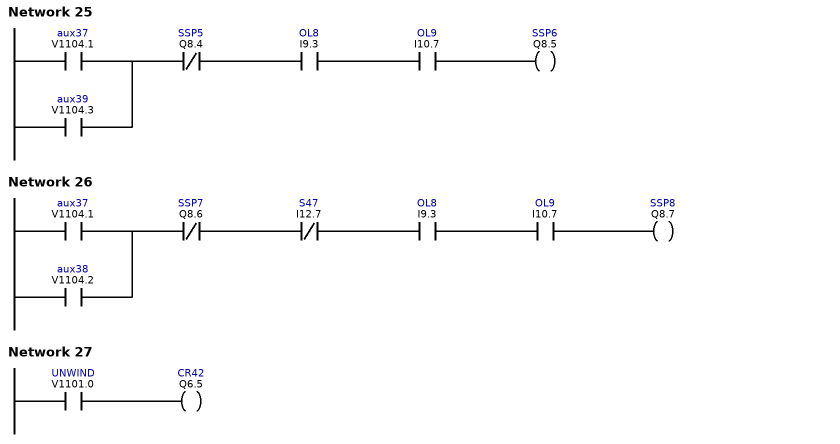
Network 25
LD     aux37:V1104.1
O      aux39:V1104.3
AN     SSP5:Q8.4
A      OL8:I9.3
A      OL9:I10.7
=      SSP6:Q8.5
Network 26
LD     aux37:V1104.1
O      aux38:V1104.2
AN     SSP7:Q8.6
AN     S47:I12.7
A      OL8:I9.3
A      OL9:I10.7
=      SSP8:Q8.7
Network 27
LD     UNWIND:V1101.0
=      CR42:Q6.5
END_SUBROUTINE_BLOCK

SUBROUTINE_BLOCK Roll_Eiector:SBR7
TITLE= SUBROUTINE COMMENTS
// Press F1 for help and example program
BEGIN
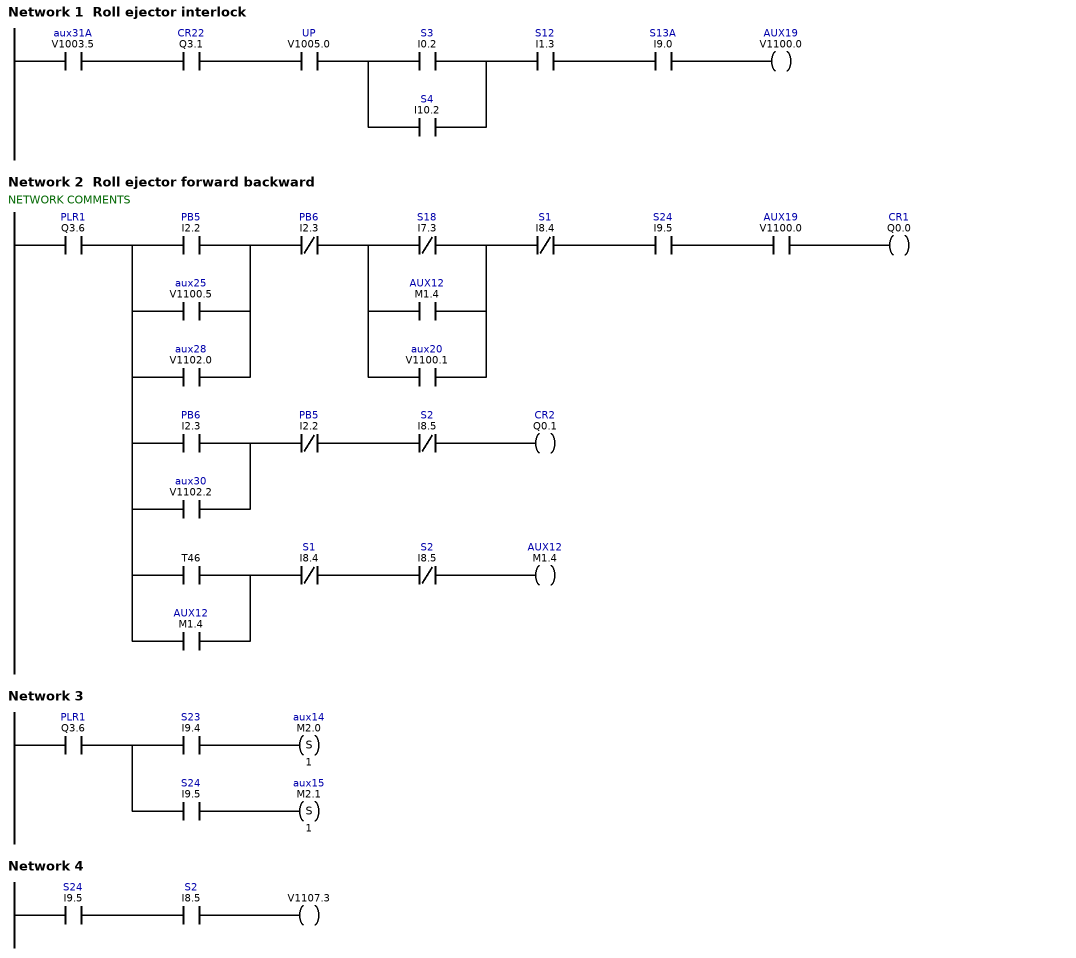
Network 1 // Roll ejector interlock
LD     aux31A:V1003.5
A      CR22:Q3.1
A      UP:V1005.0
LD     S3:I0.2
O      S4:I10.2
ALD
A      S12:I1.3
A      S13A:I9.0
=      AUX19:V1100.0
Network 2 // Roll ejector forward backward
//  NETWORK COMMENTS
LD     PLR1:Q3.6
LPS
LD     PB5:I2.2
O      aux25:V1100.5
O      aux28:V1102.0
AN     PB6:I2.3
LDN    S18:I7.3
O      AUX12:M1.4
O      aux20:V1100.1
ALD
ALD
AN     S1:I8.4
A      S24:I9.5
A      AUX19:V1100.0
=      CR1:Q0.0
LRD
LD     PB6:I2.3
O      aux30:V1102.2
ALD
AN     PB5:I2.2
AN     S2:I8.5
=      CR2:Q0.1
LPP
LD     T46
O      AUX12:M1.4
ALD
AN     S1:I8.4
AN     S2:I8.5
=      AUX12:M1.4
Network 3
LD     PLR1:Q3.6
LPS
A      S23:I9.4
S      aux14:M2.0, 1
LPP
A      S24:I9.5
S      aux15:M2.1, 1
Network 4
LD     S24:I9.5
A      S2:I8.5
=      V1107.3
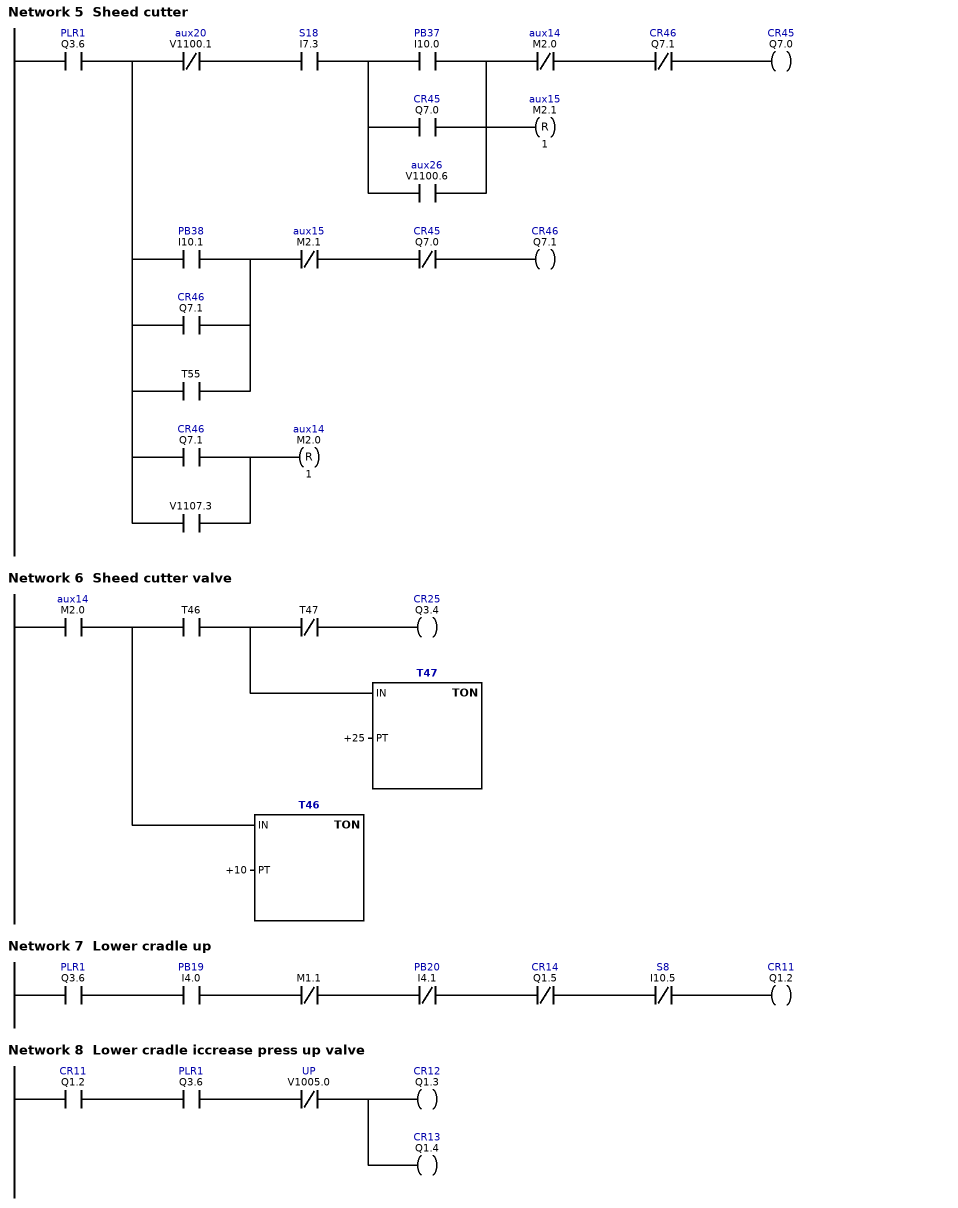
Network 5 // Sheed cutter
LD     PLR1:Q3.6
LPS
AN     aux20:V1100.1
A      S18:I7.3
LD     PB37:I10.0
O      CR45:Q7.0
O      aux26:V1100.6
ALD
LPS
AN     aux14:M2.0
AN     CR46:Q7.1
=      CR45:Q7.0
LPP
R      aux15:M2.1, 1
LRD
LD     PB38:I10.1
O      CR46:Q7.1
O      T55
ALD
AN     aux15:M2.1
AN     CR45:Q7.0
=      CR46:Q7.1
LPP
LD     CR46:Q7.1
O      V1107.3
ALD
R      aux14:M2.0, 1
Network 6 // Sheed cutter valve
LD     aux14:M2.0
LPS
A      T46
LPS
AN     T47
=      CR25:Q3.4
LPP
TON    T47, +25
LPP
TON    T46, +10
Network 7 // Lower cradle up
LD     PLR1:Q3.6
A      PB19:I4.0
AN     M1.1
AN     PB20:I4.1
AN     CR14:Q1.5
AN     S8:I10.5
=      CR11:Q1.2
Network 8 // Lower cradle iccrease press up valve
LD     CR11:Q1.2
A      PLR1:Q3.6
AN     UP:V1005.0
=      CR12:Q1.3
=      CR13:Q1.4
